// TIA Portal V18 export
TYPE "TM_Pulse_2x24_In"
   STRUCT
      Ch0 { S7_SetPoint := 'True'} : "TM_Pulse_2x24_In_PWM";
      Ch1 { S7_SetPoint := 'True'} : "TM_Pulse_2x24_In_PWM";
   END_STRUCT;
END_TYPE
